ABB RAPID module: Module1.mod

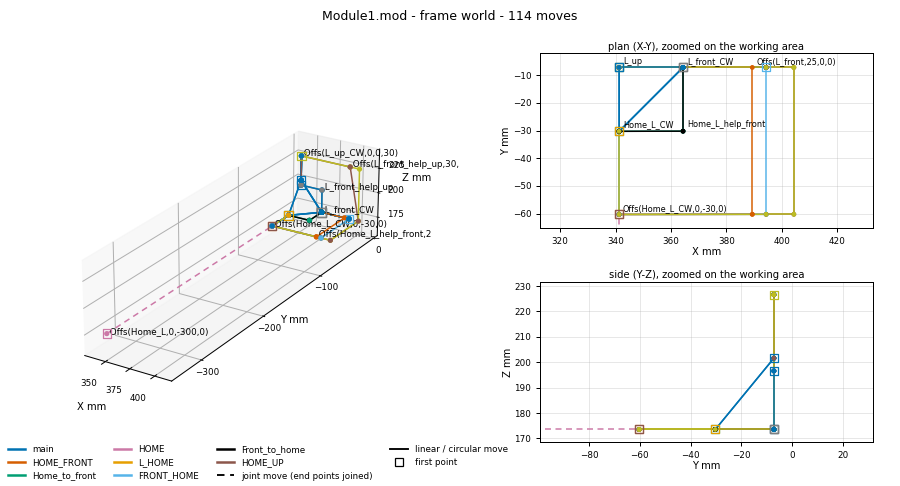
[picture p0: tool path of Module1.mod in frame world, 114 of 114 moves have a stored position in this frame; points joined in program order, loops and branches not executed]
MODULE Module1
        CONST robtarget Home_L:=[[341.275,-30.28,173.537],[0.707106781,-0.707106781,0,0],[1,-1,2,4],[-101.964427132,9E+09,9E+09,9E+09,9E+09,9E+09]];
    CONST robtarget Home_L_help_front:=[[364.325,-30.23,173.537],[0.707106781,-0.707106781,0,0],[1,-1,2,4],[-101.964427132,9E+09,9E+09,9E+09,9E+09,9E+09]];
    CONST robtarget L_front_help_home:=[[364.325,-30.23,173.537],[0.707106781,0,-0.707106781,0],[1,-1,2,4],[-101.96443282,9E+09,9E+09,9E+09,9E+09,9E+09]];
    CONST robtarget L_front:=[[364.325,-7.23,173.537],[0.707106781,0,-0.707106781,0],[1,-1,2,4],[-101.96443282,9E+09,9E+09,9E+09,9E+09,9E+09]];
    CONST robtarget L_front_help_up:=[[364.325,-7.23,196.537],[0.5,-0.5,-0.5,0.5],[1,-1,2,4],[-101.96443282,9E+09,9E+09,9E+09,9E+09,9E+09]];
    CONST robtarget L_up_from_front_help:=[[364.324659724,-7.23,196.536776157],[0,0,1,0],[1,-2,0,4],[-101.964427132,9E+09,9E+09,9E+09,9E+09,9E+09]];
    CONST robtarget L_up:=[[341.274659724,-7.23,196.586776157],[0,0,1,0],[1,-2,1,4],[-101.964427132,9E+09,9E+09,9E+09,9E+09,9E+09]];
    CONST robtarget L_front_ACW:=[[364.325,-7.23,173.537],[0.5,0.5,-0.5,-0.5],[1,-1,2,4],[-101.96443282,9E+09,9E+09,9E+09,9E+09,9E+09]];
    CONST robtarget L_front_CW:=[[364.325,-7.23,173.537],[0.5,-0.5,-0.5,0.5],[1,-1,-1,4],[-101.96443282,9E+09,9E+09,9E+09,9E+09,9E+09]];
    CONST robtarget Home_L_CW:=[[341.275,-30.28,173.537],[0.5,-0.5,0.5,0.5],[1,-1,2,4],[-101.964427132,9E+09,9E+09,9E+09,9E+09,9E+09]];
    CONST robtarget Home_L_ACW:=[[341.275,-30.28,173.537],[0.5,-0.5,-0.5,-0.5],[1,-1,2,4],[-101.964427132,9E+09,9E+09,9E+09,9E+09,9E+09]];
    CONST robtarget L_up_ACW:=[[341.274659724,-7.23,196.586776157],[0,-0.707106781,0.707106781,0],[1,-2,1,4],[-101.964427132,9E+09,9E+09,9E+09,9E+09,9E+09]];
    CONST robtarget L_up_CW:=[[341.274659724,-7.23,196.586776157],[0,0.707106781,0.707106781,0],[1,-2,1,4],[-101.964427132,9E+09,9E+09,9E+09,9E+09,9E+09]];

    !####################################### OBSLUHUJU U F L
    PROC main()
!        HOME;
!        MoveL Home_L_CW,v150,fine,Servo;
!        MoveL Home_L,v150,fine,Servo;
!        MoveL Home_L_ACW,v150,fine,Servo;
!        MoveL Home_L,v150,fine,Servo;
!        HOME_FRONT;
!        MoveL L_front_ACW,v150,fine,Servo;
!        MoveL L_front,v150,fine,Servo;
!        MoveL L_front_CW,v150,fine,Servo;
!        MoveL L_front,v150,fine,Servo;
!        FRONT_UP;
!        MoveL Offs(L_up_ACW,0,0,5),v150,fine,Servo;
!        MoveL Offs(L_up,0,0,5),v150,fine,Servo;
!        MoveL Offs(L_up_CW,0,0,5),v150,fine,Servo;
!        MoveL Offs(L_up,0,0,5),v150,fine,Servo;
!        UP_FRONT;
!        MoveL L_front_ACW,v150,fine,Servo;
!        MoveL L_front,v150,fine,Servo;
!        MoveL L_front_CW,v150,fine,Servo;
!        MoveL L_front,v150,fine,Servo;
!        FRONT_HOME;
!        MoveL Home_L_CW,v150,fine,Servo;
!        MoveL Home_L,v150,fine,Servo;
!        MoveL Home_L_ACW,v150,fine,Servo;
!        MoveL Home_L,v150,fine,Servo;
        VAR num SizeOfInputArray:=6;
        VAR string input_array{6};
        !input_array:= ["F","F'","F2","F2","R","R'","R2","R2","U","U'","U2","U2","B","B'","B2","B2","L","L'","L2","L2","D","D'","D2","D2","BREAK"];
        input_array:= ["B'","L'","D'","B'","D'","BREAK"];

        g_Init \maxSpd:=10 \holdForce:=5 \Calibrate;
        g_GripIn;!g_GripIn
        g_GripOut;

        SetDO DO_R_in_pos,1;
        WaitDO DO_L_in_pos,1;
        WaitTime 1;
        SetDO DO_R_in_pos,0;

        g_GripOut;
        WaitTime 5;
        HOME;
        WaitTime 10;
        g_GripIn;
        WaitTime 0.25;
        PulseDO DO_ATTACH_2_GL;
        WaitTime 0.25;
        SetDO DO_R_in_pos,1;
        WaitDO DO_L_in_pos,1;
        WaitTime .5;
        SetDO DO_R_in_pos,0;

      FOR i FROM 1 TO SizeOfInputArray DO
        WaitDI DI_R_in_pos,0;
        WaitDO DO_L_in_pos,0;
        TEST input_array{i}
            CASE "U" :      !cekej signal####################
                WaitDO DO_L_in_pos,1;
                g_GripOut;
                WaitTime 0.25;
                PulseDO DO_DETACH_GL;
                WaitTime 0.25;
                HOME_UP;
                g_GripIn;
                WaitTime 0.25;
                PulseDO DO_ATTACH_6_GL;
                WaitTime 0.25;
                MoveL Offs(L_up_CW,0,0,5),v150,fine,Servo;
                g_GripOut;
                WaitTime 0.25;
                PulseDO DO_DETACH_GL;
                WaitTime 0.25;
                MoveL Offs(L_up_CW,0,0,30),v150,fine,Servo;
                MoveL Offs(L_up,0,0,30),v150,fine,Servo;
                MoveL Offs(L_up,0,0,5),v150,fine,Servo;
                UP_HOME;
                g_GripIn;
                WaitTime 0.25;
                PulseDO DO_ATTACH_2_GL;
                WaitTime 0.25;
                SetDO DO_R_in_pos,1;
                WaitDO DO_L_in_pos,0;
                SetDO DO_R_in_pos,0;
            CASE "F" :      !cekej signal####################
                WaitDO DO_L_in_pos,1;
                g_GripOut;
                WaitTime 0.25;
                PulseDO DO_DETACH_GL;
                WaitTime 0.25;
                HOME_FRONT;
                g_GripIn;
                WaitTime 0.25;
                PulseDO DO_ATTACH_1_GL;
                WaitTime 0.25;
                MoveL L_front_CW,v150,fine,Servo;
                g_GripOut;
                WaitTime 0.25;
                PulseDO DO_DETACH_GL;
                WaitTime 0.25;
                MoveL Offs(L_front_CW,30,0,0),v150,fine,Servo;
                MoveL Offs(L_front,30,0,0),v150,fine,Servo;
                MoveL L_front,v150,fine,Servo;
                FRONT_HOME;
                g_GripIn;
                WaitTime 0.25;
                PulseDO DO_ATTACH_2_GL;
                WaitTime 0.25;
                SetDO DO_R_in_pos,1;
                WaitDO DO_L_in_pos,0;
                SetDO DO_R_in_pos,0;
            CASE "B" :      !NENENENEcekej signal####################
                g_GripOut;
                WaitTime 0.25;
                PulseDO DO_DETACH_GL;
                WaitTime 0.25;
                HOME_FRONT;
                g_GripIn;
                WaitTime 0.25;
                PulseDO DO_ATTACH_1_GL;
                WaitTime 0.25;
                SetDO DO_R_in_pos,1;
                WaitDO DO_L_in_pos,1;
                g_GripOut;
                WaitTime 0.25;
                PulseDO DO_DETACH_GL;
                WaitTime 0.25;
                FRONT_HOME;
                g_GripIn;
                WaitTime 0.25;
                PulseDO DO_ATTACH_2_GL;
                WaitTime 0.25;
                SetDO DO_R_in_pos,0;
            CASE "L" :      !cekej signal####################
!                WaitDO DO_L_in_pos,1;
!                g_GripOut;
!                HOME;
!                g_GripIn;
                MoveL Home_L_CW,v150,fine,Servo;
                g_GripOut;
                WaitTime 0.25;
                PulseDO DO_DETACH_GL;
                WaitTime 0.25;
                MoveL Offs(Home_L_CW,0,-30,0),v150,fine,Servo;
                MoveL Offs(Home_L,0,-30,0),v150,fine,Servo;
                MoveL Home_L,v150,fine,Servo;
!                HOME;
                g_GripIn;
                WaitTime 0.25;
                PulseDO DO_ATTACH_2_GL;
                WaitTime 0.25;
!                SetDO DO_R_in_pos,1;
!                WaitDO DO_L_in_pos,0;
!                SetDO DO_R_in_pos,0;
            CASE "R" :      !NENENENEcekej signal####################
!                g_GripOut;
!                HOME;
!                g_GripIn;
!                SetDO DO_R_in_pos,1;
!                WaitDO DO_L_in_pos,1;
!                g_GripOut;
!                HOME;
!                g_GripIn;
!                SetDO DO_R_in_pos,0;
            CASE "D" :      !NENENENEcekej signal####################
                g_GripOut;
                WaitTime 0.25;
                PulseDO DO_DETACH_GL;
                WaitTime 0.25;
                HOME_UP;
                g_GripIn;
                WaitTime 0.25;
                PulseDO DO_ATTACH_6_GL;
                WaitTime 0.25;
                SetDO DO_R_in_pos,1;
                WaitDO DO_L_in_pos,1;
                g_GripOut;
                WaitTime 0.25;
                PulseDO DO_DETACH_GL;
                WaitTime 0.25;
                UP_HOME;
                g_GripIn;
                WaitTime 0.25;
                PulseDO DO_ATTACH_2_GL;
                WaitTime 0.25;
                SetDO DO_R_in_pos,0;
            CASE "U2" :
                WaitDO DO_L_in_pos,1;
                g_GripOut;
                WaitTime 0.25;
                PulseDO DO_DETACH_GL;
                WaitTime 0.25;
                HOME_UP;
                g_GripIn;
                WaitTime 0.25;
                PulseDO DO_ATTACH_6_GL;
                WaitTime 0.25;
                MoveL Offs(L_up_CW,0,0,5),v150,fine,Servo;
                g_GripOut;
                WaitTime 0.25;
                PulseDO DO_DETACH_GL;
                WaitTime 0.25;
                MoveL Offs(L_up_CW,0,0,30),v150,fine,Servo;
                MoveL Offs(L_up,0,0,30),v150,fine,Servo;
                MoveL Offs(L_up,0,0,5),v150,fine,Servo;
                g_GripIn;
                WaitTime 0.25;
                PulseDO DO_ATTACH_6_GL;
                WaitTime 0.25;
                MoveL Offs(L_up_CW,0,0,5),v150,fine,Servo;
                g_GripOut;
                WaitTime 0.25;
                PulseDO DO_DETACH_GL;
                WaitTime 0.25;
                MoveL Offs(L_up_CW,0,0,30),v150,fine,Servo;
                MoveL Offs(L_up,0,0,30),v150,fine,Servo;
                MoveL Offs(L_up,0,0,5),v150,fine,Servo;
                UP_HOME;
                g_GripIn;
                WaitTime 0.25;
                PulseDO DO_ATTACH_2_GL;
                WaitTime 0.25;
                SetDO DO_R_in_pos,1;
                WaitDO DO_L_in_pos,0;
                SetDO DO_R_in_pos,0;
            CASE "F2" :
                WaitDO DO_L_in_pos,1;
                g_GripOut;
                WaitTime 0.25;
                PulseDO DO_DETACH_GL;
                WaitTime 0.25;
                HOME_FRONT;
                g_GripIn;
                WaitTime 0.25;
                PulseDO DO_ATTACH_1_GL;
                WaitTime 0.25;
                MoveL L_front_CW,v150,fine,Servo;
                g_GripOut;
                WaitTime 0.25;
                PulseDO DO_DETACH_GL;
                WaitTime 0.25;
                MoveL Offs(L_front_CW,30,0,0),v150,fine,Servo;
                MoveL Offs(L_front,30,0,0),v150,fine,Servo;
                MoveL L_front,v150,fine,Servo;
                g_GripIn;
                WaitTime 0.25;
                PulseDO DO_ATTACH_1_GL;
                WaitTime 0.25;
                MoveL L_front_CW,v150,fine,Servo;
                g_GripOut;
                WaitTime 0.25;
                PulseDO DO_DETACH_GL;
                WaitTime 0.25;
                MoveL Offs(L_front_CW,30,0,0),v150,fine,Servo;
                MoveL Offs(L_front,30,0,0),v150,fine,Servo;
                MoveL L_front,v150,fine,Servo;
                FRONT_HOME;
                g_GripIn;
                WaitTime 0.25;
                PulseDO DO_ATTACH_2_GL;
                WaitTime 0.25;
                SetDO DO_R_in_pos,1;
                WaitDO DO_L_in_pos,0;
                SetDO DO_R_in_pos,0;
            CASE "B2" :
                g_GripOut;
                WaitTime 0.25;
                PulseDO DO_DETACH_GL;
                WaitTime 0.25;
                HOME_FRONT;
                g_GripIn;
                WaitTime 0.25;
                PulseDO DO_ATTACH_1_GL;
                WaitTime 0.25;
                SetDO DO_R_in_pos,1;
                WaitDO DO_L_in_pos,1;
                g_GripOut;
                WaitTime 0.25;
                PulseDO DO_DETACH_GL;
                WaitTime 0.25;
                FRONT_HOME;
                g_GripIn;
                WaitTime 0.25;
                PulseDO DO_ATTACH_2_GL;
                WaitTime 0.25;
                SetDO DO_R_in_pos,0;
            CASE "L2" :
!                WaitDO DO_L_in_pos,1;
!                g_GripOut;
!                HOME;
!                g_GripIn;
                MoveL Home_L_CW,v150,fine,Servo;
                g_GripOut;
                WaitTime 0.25;
                PulseDO DO_DETACH_GL;
                WaitTime 0.25;
                MoveL Offs(Home_L_CW,0,-30,0),v150,fine,Servo;
                MoveL Offs(Home_L,0,-30,0),v150,fine,Servo;
                MoveL Home_L,v150,fine,Servo;
!                HOME;
                g_GripIn;
                WaitTime 0.25;
                PulseDO DO_ATTACH_2_GL;
                WaitTime 0.25;
                MoveL Home_L_CW,v150,fine,Servo;
                g_GripOut;
                WaitTime 0.25;
                PulseDO DO_DETACH_GL;
                WaitTime 0.25;
                MoveL Offs(Home_L_CW,0,-30,0),v150,fine,Servo;
                MoveL Offs(Home_L,0,-30,0),v150,fine,Servo;
                MoveL Home_L,v150,fine,Servo;
!                HOME;
                g_GripIn;
                WaitTime 0.25;
                PulseDO DO_ATTACH_2_GL;
                WaitTime 0.25;
!                SetDO DO_R_in_pos,1;
!                WaitDO DO_L_in_pos,0;
!                SetDO DO_R_in_pos,0;
            CASE "R2" :
!                g_GripOut;
!                HOME;
!                g_GripIn;
!                SetDO DO_R_in_pos,1;
!                WaitDO DO_L_in_pos,1;
!                g_GripOut;
!                HOME;
!                g_GripIn;
!                SetDO DO_R_in_pos,0;
            CASE "D2" :
                g_GripOut;
                WaitTime 0.25;
                PulseDO DO_DETACH_GL;
                WaitTime 0.25;
                HOME_UP;
                g_GripIn;
                WaitTime 0.25;
                PulseDO DO_ATTACH_6_GL;
                WaitTime 0.25;
                SetDO DO_R_in_pos,1;
                WaitDO DO_L_in_pos,1;
                g_GripOut;
                WaitTime 0.25;
                PulseDO DO_DETACH_GL;
                WaitTime 0.25;
                UP_HOME;
                g_GripIn;
                WaitTime 0.25;
                PulseDO DO_ATTACH_2_GL;
                WaitTime 0.25;
                SetDO DO_R_in_pos,0;
            CASE "U'" :
                WaitDO DO_L_in_pos,1;
                g_GripOut;
                WaitTime 0.25;
                PulseDO DO_DETACH_GL;
                WaitTime 0.25;
                HOME_UP;
                g_GripIn;
                WaitTime 0.25;
                PulseDO DO_ATTACH_6_GL;
                WaitTime 0.25;
                MoveL Offs(L_up_ACW,0,0,5),v150,fine,Servo;
                g_GripOut;
                WaitTime 0.25;
                PulseDO DO_DETACH_GL;
                WaitTime 0.25;
                MoveL Offs(L_up_ACW,0,0,30),v150,fine,Servo;
                MoveL Offs(L_up,0,0,30),v150,fine,Servo;
                MoveL Offs(L_up,0,0,5),v150,fine,Servo;
                UP_HOME;
                g_GripIn;
                WaitTime 0.25;
                PulseDO DO_ATTACH_2_GL;
                WaitTime 0.25;
                SetDO DO_R_in_pos,1;
                WaitDO DO_L_in_pos,0;
                SetDO DO_R_in_pos,0;
            CASE "F'" :
                WaitDO DO_L_in_pos,1;
                g_GripOut;
                WaitTime 0.25;
                PulseDO DO_DETACH_GL;
                WaitTime 0.25;
                HOME_FRONT;
                g_GripIn;
                WaitTime 0.25;
                PulseDO DO_ATTACH_1_GL;
                WaitTime 0.25;
                MoveL L_front_ACW,v150,fine,Servo;
                g_GripOut;
                WaitTime 0.25;
                PulseDO DO_DETACH_GL;
                WaitTime 0.25;
                MoveL Offs(L_front_ACW,30,0,0),v150,fine,Servo;
                MoveL Offs(L_front,30,0,0),v150,fine,Servo;
                MoveL L_front,v150,fine,Servo;
                FRONT_HOME;
                g_GripIn;
                WaitTime 0.25;
                PulseDO DO_ATTACH_2_GL;
                WaitTime 0.25;
                SetDO DO_R_in_pos,1;
                WaitDO DO_L_in_pos,0;
                SetDO DO_R_in_pos,0;
            CASE "B'" :
                g_GripOut;
                WaitTime 0.25;
                PulseDO DO_DETACH_GL;
                WaitTime 0.25;
                HOME_FRONT;
                g_GripIn;
                WaitTime 0.25;
                PulseDO DO_ATTACH_1_GL;
                WaitTime 0.25;
                SetDO DO_R_in_pos,1;
                WaitDO DO_L_in_pos,1;
                g_GripOut;
                WaitTime 0.25;
                PulseDO DO_DETACH_GL;
                WaitTime 0.25;
                FRONT_HOME;
                g_GripIn;
                WaitTime 0.25;
                PulseDO DO_ATTACH_2_GL;
                WaitTime 0.25;
                SetDO DO_R_in_pos,0;
            CASE "L'" :
!                WaitDO DO_L_in_pos,1;
!                g_GripOut;
!                HOME;
!                g_GripIn;
                MoveL Home_L_ACW,v150,fine,Servo;
                g_GripOut;
                WaitTime 0.25;
                PulseDO DO_DETACH_GL;
                WaitTime 0.25;
                MoveL Offs(Home_L_ACW,0,-30,0),v150,fine,Servo;
                MoveL Offs(Home_L,0,-30,0),v150,fine,Servo;
                MoveL Home_L,v150,fine,Servo;
!                HOME;
                g_GripIn;
                WaitTime 0.25;
                PulseDO DO_ATTACH_2_GL;
                WaitTime 0.25;
!                SetDO DO_R_in_pos,1;
!                WaitDO DO_L_in_pos,0;
!                SetDO DO_R_in_pos,0;
            CASE "R'" :
!                g_GripOut;
!                HOME;
!                g_GripIn;
!                SetDO DO_R_in_pos,1;
!                WaitDO DO_L_in_pos,1;
!                g_GripOut;
!                HOME;
!                g_GripIn;
!                SetDO DO_R_in_pos,0;
            CASE "D'" :
                g_GripOut;
                WaitTime 0.25;
                PulseDO DO_DETACH_GL;
                WaitTime 0.25;
                HOME_UP;
                g_GripIn;
                WaitTime 0.25;
                PulseDO DO_ATTACH_6_GL;
                WaitTime 0.25;
                SetDO DO_R_in_pos,1;
                WaitDO DO_L_in_pos,1;
                g_GripOut;
                WaitTime 0.25;
                PulseDO DO_DETACH_GL;
                WaitTime 0.25;
                UP_HOME;
                g_GripIn;
                WaitTime 0.25;
                PulseDO DO_ATTACH_2_GL;
                WaitTime 0.25;
                SetDO DO_R_in_pos,0;
            CASE "BREAK" :
                BREAK;
        ENDTEST

      ENDFOR

        !Add your code here
    ENDPROC
    PROC HOME_FRONT()
        MoveL Offs(Home_L,0,-30,0),v150,fine,Servo;
        MoveL Offs(Home_L_help_front,25,-30,0),v150,fine,Servo;
        MoveL Offs(L_front_help_home,25,-30,0),v150,fine,Servo;
        MoveL Offs(L_front,25,0,0),v150,fine,Servo;
        MoveL L_front,v150,fine,Servo;
    ENDPROC
    PROC Home_to_front()
        MoveL Home_L,v150,fine,Servo\WObj:=wobj0;
        MoveL Home_L_help_front,v150,fine,Servo\WObj:=wobj0;
        MoveL L_front_help_home,v150,fine,Servo\WObj:=wobj0;
        MoveL L_front,v150,fine,Servo\WObj:=wobj0;
        MoveL L_front_ACW,v150,fine,Servo\WObj:=wobj0;
        MoveL L_front,v150,fine,Servo\WObj:=wobj0;
        MoveL L_front_CW,v150,fine,Servo\WObj:=wobj0;
        MoveL L_front,v150,fine,Servo\WObj:=wobj0;
    ENDPROC
    PROC HOME()
        MoveJ Offs(Home_L,0,-300,0),v150,fine,Servo;
        MoveJ Offs(Home_L,0,-30,0),v150,fine,Servo;
        MoveL Home_L,v150,fine,Servo;
    ENDPROC
    PROC L_HOME()
        MoveJ Home_L,v150,fine,Servo\WObj:=wobj0;
        MoveL Home_L_CW,v150,fine,Servo\WObj:=wobj0;
        MoveL Home_L,v150,fine,Servo\WObj:=wobj0;
        MoveL Home_L_ACW,v150,fine,Servo\WObj:=wobj0;
        MoveL Home_L,v150,fine,Servo\WObj:=wobj0;
    ENDPROC
    PROC FRONT_HOME()
        MoveL Offs(L_front,30,0,0),v150,fine,Servo;
        MoveL Offs(L_front_help_home,30,-30,0),v150,fine,Servo;
        MoveL Offs(Home_L_help_front,30,-30,0),v150,fine,Servo;
        MoveL Offs(Home_L,0,-30,0),v150,fine,Servo;
        MoveL Home_L,v150,fine,Servo;
    ENDPROC
    PROC Front_to_home()
        MoveL L_front,v150,fine,Servo\WObj:=wobj0;
        MoveL L_front_help_home,v150,fine,Servo\WObj:=wobj0;
        MoveL Home_L_help_front,v150,fine,Servo\WObj:=wobj0;
        MoveL Home_L,v150,fine,Servo\WObj:=wobj0;
        MoveL Home_L_ACW,v150,fine,Servo\WObj:=wobj0;
        MoveL Home_L,v150,fine,Servo\WObj:=wobj0;
        MoveL Home_L_CW,v150,fine,Servo\WObj:=wobj0;
        MoveL Home_L,v150,fine,Servo\WObj:=wobj0;
    ENDPROC
    PROC HOME_UP()
        MoveL Offs(Home_L,0,-30,0),v150,fine,Servo;
        MoveL Offs(Home_L_help_front,30,-30,0),v150,fine,Servo;
        MoveL Offs(L_front_help_home,40,-30,0),v150,fine,Servo;
        MoveL Offs(L_front,40,0,0),v150,fine,Servo;
        MoveL Offs(L_front_help_up,30,0,30),v150,fine,Servo;
        MoveL Offs(L_up_from_front_help,30,0,30),v150,fine,Servo;
        MoveL Offs(L_up,0,0,30),v150,fine,Servo;
        MoveL Offs(L_up,0,0,5),v150,fine,Servo;
    ENDPROC
    PROC Front_to_up()
        MoveL L_front,v150,fine,Servo\WObj:=wobj0;
        MoveL L_front_help_up,v150,fine,Servo\WObj:=wobj0;
        MoveL L_up_from_front_help,v150,fine,Servo\WObj:=wobj0;
        MoveL L_up,v150,fine,Servo\WObj:=wobj0;
        MoveL L_up_ACW,v150,fine,Servo\WObj:=wobj0;
        MoveL L_up,v150,fine,Servo\WObj:=wobj0;
        MoveL L_up_CW,v150,fine,Servo\WObj:=wobj0;
        MoveL L_up,v150,fine,Servo\WObj:=wobj0;
    ENDPROC
    PROC UP_HOME()
        MoveL Offs(L_up,0,0,30),v150,fine,Servo;
        MoveL Offs(L_up_from_front_help,30,0,30),v150,fine,Servo;
        MoveL Offs(L_front_help_up,40,0,30),v150,fine,Servo;
        MoveL Offs(L_front,40,0,0),v150,fine,Servo;
        MoveL Offs(L_front_help_home,40,-30,0),v150,fine,Servo;
        MoveL Offs(Home_L_help_front,30,-30,0),v150,fine,Servo;
        MoveL Offs(Home_L,0,-30,0),v150,fine,Servo;
        MoveL Home_L,v150,fine,Servo;
    ENDPROC
    PROC Up_to_front()
        MoveL L_up,v150,fine,Servo\WObj:=wobj0;
        MoveL L_up_from_front_help,v150,fine,Servo\WObj:=wobj0;
        MoveL L_front_help_up,v150,fine,Servo\WObj:=wobj0;
        MoveL L_front,v150,fine,Servo\WObj:=wobj0;
        MoveL L_front_CW,v150,fine,Servo\WObj:=wobj0;
        MoveL L_front,v150,fine,Servo\WObj:=wobj0;
        MoveL L_front_ACW,v150,fine,Servo\WObj:=wobj0;
        MoveL L_front,v150,fine,Servo\WObj:=wobj0;
    ENDPROC
ENDMODULE
